// TIA Portal V19 export
FUNCTION "DEBUG_Check_Fun_Msg_100" : Void   // FC201, LAD
// stored: SetENOAutomatically false
   VAR_TEMP   // added for the SCL form of the ladder/FBD networks
      _w1 : Bool;
   END_VAR
BEGIN

REGION Network 1
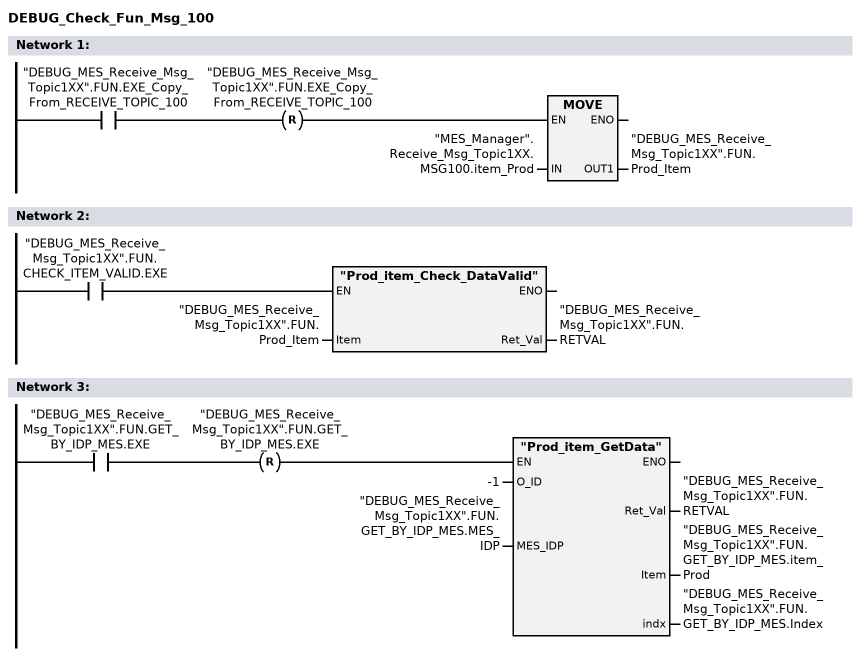
   RUNG wire#powerrail
      Contact( "DEBUG_MES_Receive_Msg_Topic1XX".FUN.EXE_Copy_From_RECEIVE_TOPIC_100 )
      R_Coil( "DEBUG_MES_Receive_Msg_Topic1XX".FUN.EXE_Copy_From_RECEIVE_TOPIC_100 )
      Move(in := "MES_Manager".Receive_Msg_Topic1XX.MSG100.item_Prod, out1 => "DEBUG_MES_Receive_Msg_Topic1XX".FUN.Prod_Item)
   END_RUNG
   // the same network as SCL:
   #_w1 := "DEBUG_MES_Receive_Msg_Topic1XX".FUN.EXE_Copy_From_RECEIVE_TOPIC_100;
   IF #_w1 THEN
       "DEBUG_MES_Receive_Msg_Topic1XX".FUN.EXE_Copy_From_RECEIVE_TOPIC_100 := FALSE;
       "DEBUG_MES_Receive_Msg_Topic1XX".FUN.Prod_Item := "MES_Manager".Receive_Msg_Topic1XX.MSG100.item_Prod;
   END_IF;
END_REGION

REGION Network 2
   RUNG wire#powerrail
      Contact( "DEBUG_MES_Receive_Msg_Topic1XX".FUN.CHECK_ITEM_VALID.EXE )
      "Prod_item_Check_DataValid"(Item := "DEBUG_MES_Receive_Msg_Topic1XX".FUN.Prod_Item, Ret_Val => "DEBUG_MES_Receive_Msg_Topic1XX".FUN.RETVAL)
   END_RUNG
   // the same network as SCL:
   IF "DEBUG_MES_Receive_Msg_Topic1XX".FUN.CHECK_ITEM_VALID.EXE THEN
       "DEBUG_MES_Receive_Msg_Topic1XX".FUN.RETVAL := "Prod_item_Check_DataValid"(Item := "DEBUG_MES_Receive_Msg_Topic1XX".FUN.Prod_Item);
   END_IF;
END_REGION

REGION Network 3
   RUNG wire#powerrail
      Contact( "DEBUG_MES_Receive_Msg_Topic1XX".FUN.GET_BY_IDP_MES.EXE )
      R_Coil( "DEBUG_MES_Receive_Msg_Topic1XX".FUN.GET_BY_IDP_MES.EXE )
      "Prod_item_GetData"(O_ID := -1, MES_IDP := "DEBUG_MES_Receive_Msg_Topic1XX".FUN.GET_BY_IDP_MES.MES_IDP, Ret_Val => "DEBUG_MES_Receive_Msg_Topic1XX".FUN.RETVAL, Item => "DEBUG_MES_Receive_Msg_Topic1XX".FUN.GET_BY_IDP_MES.item_Prod, indx => "DEBUG_MES_Receive_Msg_Topic1XX".FUN.GET_BY_IDP_MES.Index)
   END_RUNG
   // the same network as SCL:
   #_w1 := "DEBUG_MES_Receive_Msg_Topic1XX".FUN.GET_BY_IDP_MES.EXE;
   IF #_w1 THEN
       "DEBUG_MES_Receive_Msg_Topic1XX".FUN.GET_BY_IDP_MES.EXE := FALSE;
       "DEBUG_MES_Receive_Msg_Topic1XX".FUN.RETVAL := "Prod_item_GetData"(O_ID := -1,
                               MES_IDP := "DEBUG_MES_Receive_Msg_Topic1XX".FUN.GET_BY_IDP_MES.MES_IDP,
                               Item => "DEBUG_MES_Receive_Msg_Topic1XX".FUN.GET_BY_IDP_MES.item_Prod,
                               indx => "DEBUG_MES_Receive_Msg_Topic1XX".FUN.GET_BY_IDP_MES.Index);
   END_IF;
END_REGION
END_FUNCTION
